TYPE HMI_SP_TemplateClean :
STRUCT
	MachinePartEnabled:BOOL:=TRUE;				//block is enabled >> can be used to disable part(s) of the machine
END_STRUCT
END_TYPE

(* stored: Version 1.1.0.1
   DUT HMI_SP_TemplateClean: Id {fa7b424d-320a-46fe-aa94-64457783369a} *)
